Staubli VAL3: pauseCycle.pgx

public program pauseCycle()
begin
  // pause the cycle
  if !cycleStatus:bPause
    logMsg("[KERNEL] CYCLE:Pause the cycle")
    // pause the robot
    cycleStatus:bToPause=true
    watch(cycleStatus:bToPause==false,1)
  endIf
end
